//{attribute 'qualified_only'}
//{attribute 'strict'}
TYPE E_MessageList :
(
	eNO_MESSAGE := 0,
	eDEBUG_MESSAGE,
	eVON_DRUCKTISCH_UEBERNOMMEN,
	eAN_DRUCKTISCH_UEBERGEBEN,
	eVON_UMLENKUNG_UEBERNOMMER,
	eAN_UMLENKUNG_UEBERGEBEN,
	eAN_SCHNEIDEN_UEBERGEN,
	eCONVEYOR_1_AT_TRANSFER_POINT,
	eCONVEYOR_1_RESUMING_OPERATION,
	eCONVEYOR_2_AT_TRANSFER_POINT,
	eCONVEYOR_2_RESUMING_OPERATION,
	eCONVEYOR_3_AT_TRANSFER_POINT,
	eCONVEYOR_3_RESUMING_OPERATION,
	eCONVEYOR_4_AT_TRANSFER_POINT,
	eCONVEYOR_4_RESUMING_OPERATION
)UINT;
END_TYPE

(* stored: Version 1.1.0.1, ProductVersion 3.1.4022.12
   DUT E_MessageList: Id {39c3407e-4fc3-4513-9700-64dbbdfc8b61} *)
